# EPICS autosave request: BKHOFF/iocBoot/iocBKHOFF-IOC-01/BKHOFF_01_positions.req
file "motor_positions.req" P=$(P),M=MTR$(CCP)01
file "motor_positions.req" P=$(P),M=MTR$(CCP)02
